TYPE ST_GlobalStatus :
STRUCT
	nDummy							: INT;			// Some value
END_STRUCT
END_TYPE

(* stored: Version 1.1.0.1, ProductVersion 3.1.4024.12
   DUT ST_GlobalStatus: Id {75fa6e8b-c3e6-409e-8bcc-797c9bbcaa0e} *)
